// TIA Portal V17 export
// export: Created 2021-12-03T08:13:01.9644948Z, ExportSetting WithDefaults, DisplayName Totally Integrated Automation Portal, DisplayVersion V17, DisplayName TIA Portal Openness, DisplayVersion V17, DisplayName TIA Portal Version Control Interface, DisplayVersion V17, DisplayName STEP 7 Professional, DisplayVersion V17, DisplayName STEP 7 Safety, DisplayVersion V17, DisplayName WinCC Advanced, DisplayVersion V17
FUNCTION_BLOCK "FB_MN_Acc_Ctrl"   // FB61, FBD
VERSION : 0.1
// stored: AutoNumber false, IsIECCheckEnabled true, UDAEnableTagReadback false
   VAR_INPUT
      I_InitTrue { ExternalVisible := 'False'; ExternalWritable := 'False'} : Bool;   // Инициализация
      I_Acc_PwrOnRq { ExternalVisible := 'False'; ExternalWritable := 'False'} : Bool;   // Запрос на включение
      I_AccChil_PwrIsOn { ExternalVisible := 'False'; ExternalWritable := 'False'} : Bool;   // Чиллер включен
      I_Mod220V_PwrIsOn { ExternalVisible := 'False'; ExternalWritable := 'False'} : Bool;   // Модулятор 220 В включен
      I_Mod380V_PwrIsOn { ExternalVisible := 'False'; ExternalWritable := 'False'} : Bool;   // Модулятор 380 В включен
      I_AccCS_PrwIsOn { ExternalVisible := 'False'; ExternalWritable := 'False'} : Bool;   // Ускоритель включен
      I_AccRemMode { ExternalVisible := 'False'; ExternalWritable := 'False'} : Bool;   // Удаленный режим
      I_AccWarmUp { ExternalVisible := 'False'; ExternalWritable := 'False'} : Bool;   // Прогрев ускорителя
      I_AccClear { ExternalVisible := 'False'; ExternalWritable := 'False'} : Bool;   // Предварительная готовность
      I_AccStandby { ExternalVisible := 'False'; ExternalWritable := 'False'} : Bool;   // Пауза
      I_AccReady { ExternalVisible := 'False'; ExternalWritable := 'False'} : Bool;   // Основная готовность
      I_RFOn_Rq { ExternalVisible := 'False'; ExternalWritable := 'False'} : Bool;
      I_XRay_Rq { ExternalVisible := 'False'; ExternalWritable := 'False'} : Bool;
      I_Acc_PwrOffRq { ExternalVisible := 'False'; ExternalWritable := 'False'} : Bool;   // Запрос на отключение
      I_ChillOffDly { ExternalVisible := 'False'; ExternalWritable := 'False'} : Bool;   // Чиллер включен
      I_AccFault { ExternalVisible := 'False'; ExternalWritable := 'False'} : Bool;   // Ошибка ускорителя
      I_NOEStop { ExternalVisible := 'False'; ExternalWritable := 'False'} : Bool;   // Аварийный останов
      I_FltRst { ExternalVisible := 'False'; ExternalWritable := 'False'} : Bool;   // Сигнал сбросить ошибки
      I_FullWarmUp { ExternalVisible := 'False'; ExternalWritable := 'False'} : Bool;   // Полный прогрев
      I_SafePeriIsCls { ExternalVisible := 'False'; ExternalWritable := 'False'} : Bool;   // Периметр закрыт
      I_PwrRst { ExternalVisible := 'False'; ExternalWritable := 'False'} : Bool;
   END_VAR
   VAR_OUTPUT
      O_AccPreh_PwrOn { ExternalVisible := 'False'; ExternalWritable := 'False'} : Bool;   // Включение сушки ускорителя
      O_Mod380V_RlyOn { ExternalVisible := 'False'; ExternalWritable := 'False'} : Bool;   // Включить модулятор 380 В
      O_AccMod220V_PwrOn { ExternalVisible := 'False'; ExternalWritable := 'False'} : Bool;   // Включить модулятор 220 В
      O_Chil_PwrOn { ExternalVisible := 'False'; ExternalWritable := 'False'} : Bool;   // Включить - отключть чиллер
      O_FltRst { ExternalVisible := 'False'; ExternalWritable := 'False'} : Bool;   // Сброс ошибки / Reset
      O_WarmUp { ExternalVisible := 'False'; ExternalWritable := 'False'} : Bool;   // Запрос на прогрев
      O_RFOn { ExternalVisible := 'False'; ExternalWritable := 'False'} : Bool;   // Включить СВЧ
      O_XRay_On { ExternalVisible := 'False'; ExternalWritable := 'False'} : Bool;   // Включить ТИ
      O_FullWarmUp_Rq { ExternalVisible := 'False'; ExternalWritable := 'False'} : Bool;   // Запрос на полный прогрев
      O_Acc_ActState { ExternalVisible := 'False'; ExternalWritable := 'False'} : Int;   // Состояние ускорителя
   END_VAR
   VAR DB_SPECIFIC
      S_PwrRst { ExternalVisible := 'False'} : Bool;
      AxSR { ExternalVisible := 'False'; ExternalWritable := 'False'} : Struct
         Acc230V_PwrOn { ExternalVisible := 'False'; ExternalWritable := 'False'} : Bool;
      END_STRUCT;
      S_Transit { ExternalVisible := 'False'; ExternalWritable := 'False'} : Struct
         InitTrue { ExternalVisible := 'False'; ExternalWritable := 'False'} : Bool;   // Инициализация
         ReqAccPwrOn { ExternalVisible := 'False'; ExternalWritable := 'False'} : Bool;   // Запрос на включение
         ChillOnDly { ExternalVisible := 'False'; ExternalWritable := 'False'} : Bool;   // Чиллер включен
         ModOnDly { ExternalVisible := 'False'; ExternalWritable := 'False'} : Bool;   // Модулятор включен
         AccPrwOn { ExternalVisible := 'False'; ExternalWritable := 'False'} : Bool;   // Ускоритель включен
         NAccPrwOn { ExternalVisible := 'False'; ExternalWritable := 'False'} : Bool;   // Ускоритель НЕ включен
         AccRemMode { ExternalVisible := 'False'; ExternalWritable := 'False'} : Bool;   // Удаленный режим
         NAccRemMode { ExternalVisible := 'False'; ExternalWritable := 'False'} : Bool;   // Местный режим
         AccWarmUp { ExternalVisible := 'False'; ExternalWritable := 'False'} : Bool;   // Прогрев ускорителя
         AccClear { ExternalVisible := 'False'; ExternalWritable := 'False'} : Bool;   // Предварительная готовность
         AccStandby { ExternalVisible := 'False'; ExternalWritable := 'False'} : Bool;   // Пауза
         AccReady { ExternalVisible := 'False'; ExternalWritable := 'False'} : Bool;   // Основная готовность
         AccRfOn { ExternalVisible := 'False'; ExternalWritable := 'False'} : Bool;   // СВЧ включено
         AccRfOff { ExternalVisible := 'False'; ExternalWritable := 'False'} : Bool;
         AccXrayOn { ExternalVisible := 'False'; ExternalWritable := 'False'} : Bool;   // ТИ включено
         AccXrayOff { ExternalVisible := 'False'; ExternalWritable := 'False'} : Bool;   // ТИ вЫключено
         ReqAccPwrOff { ExternalVisible := 'False'; ExternalWritable := 'False'} : Bool;   // Запрос на отключение
         AccNotActive { ExternalVisible := 'False'; ExternalWritable := 'False'} : Bool;   // Ускоритель неактивен
         XrayHeadOffDly { ExternalVisible := 'False'; ExternalWritable := 'False'} : Bool;   // Накал выключен
         ModOffDly { ExternalVisible := 'False'; ExternalWritable := 'False'} : Bool;   // Модулятор выключен
         ChillOffDly { ExternalVisible := 'False'; ExternalWritable := 'False'} : Bool;   // Чиллер включен
         AccFault { ExternalVisible := 'False'; ExternalWritable := 'False'} : Bool;   // Ошибка ускорителя
         ACK_AccFault { ExternalVisible := 'False'; ExternalWritable := 'False'} : Bool;   // Ошибка сброшена
         EStop { ExternalVisible := 'False'; ExternalWritable := 'False'} : Bool;   // Аварийный останов
      END_STRUCT;
   END_VAR
   VAR
      DI_Acc_StateCase { ExternalVisible := 'False'; S7_SetPoint := 'True'} : "FB_Acc_StateCase";
   END_VAR
   VAR DB_SPECIFIC
      S_Acc_ActState { ExternalVisible := 'False'; ExternalWritable := 'False'} : Int;   // Состояние ускорителя
   END_VAR
   VAR_TEMP
      T_Mod230V_PwrOn : Bool;
      T_FltRst : Bool;
      T_Acc230V_PwrOn : Bool;
      T_Mod400V_PwrOn : Bool;
      T_StandBy : Bool;
      T_RFOn : Bool;
      T_XRayOn : Bool;
      T_ReqPwrOn : Bool;
   END_VAR
BEGIN

REGION Network 2: INIT / Инициализация
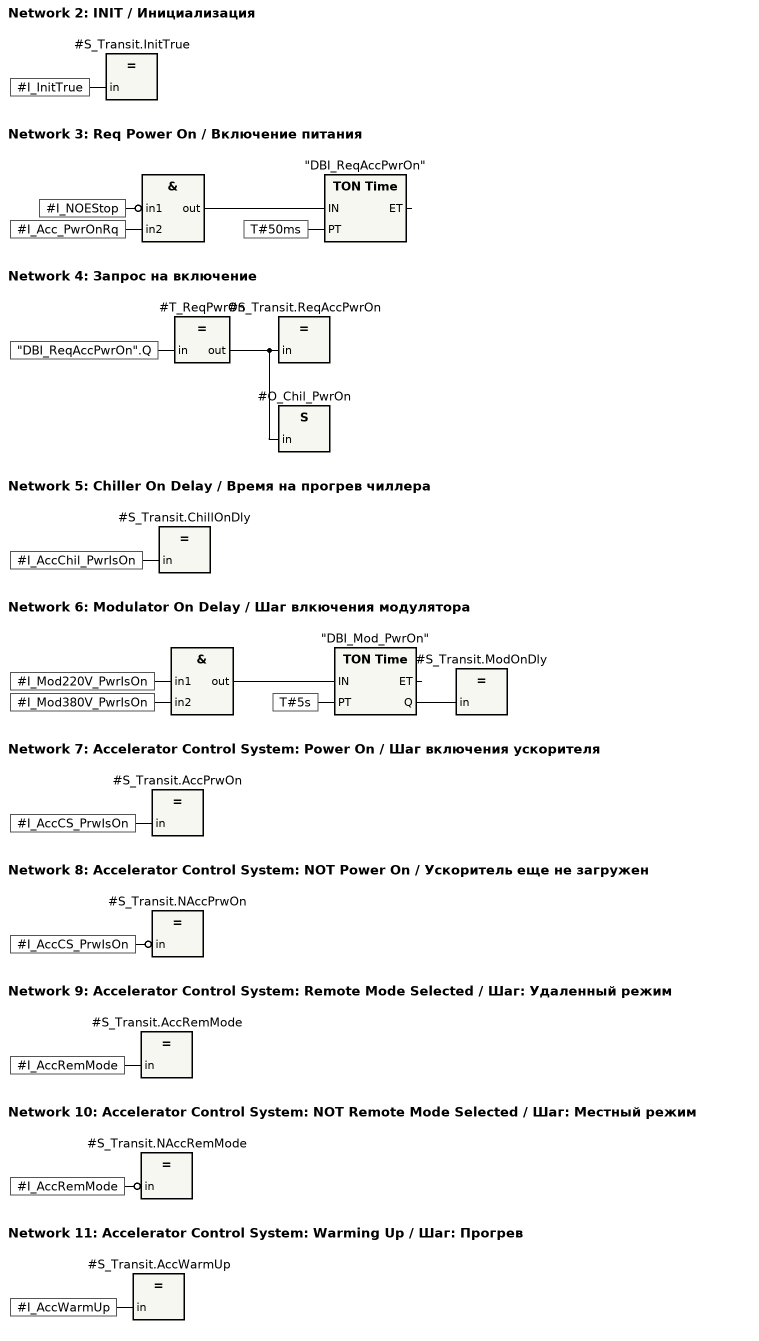
   #S_Transit.InitTrue := #I_InitTrue;
END_REGION

REGION Network 3: Req Power On / Включение питания
   "DBI_ReqAccPwrOn".TON(IN := NOT #I_NOEStop AND #I_Acc_PwrOnRq, PT := T#50ms);
END_REGION

REGION Network 4: Запрос на включение
   #T_ReqPwrOn := "DBI_ReqAccPwrOn".Q;
   #S_Transit.ReqAccPwrOn := "DBI_ReqAccPwrOn".Q;
   IF "DBI_ReqAccPwrOn".Q THEN #O_Chil_PwrOn := TRUE; END_IF;
END_REGION

REGION Network 5: Chiller On Delay / Время на прогрев чиллера
   #S_Transit.ChillOnDly := #I_AccChil_PwrIsOn;
END_REGION

REGION Network 6: Modulator On Delay / Шаг влкючения модулятора
   "DBI_Mod_PwrOn".TON(IN := #I_Mod220V_PwrIsOn AND #I_Mod380V_PwrIsOn, PT := T#5s);
   #S_Transit.ModOnDly := "DBI_Mod_PwrOn".Q;
END_REGION

REGION Network 7: Accelerator Control System: Power On / Шаг включения ускорителя
   #S_Transit.AccPrwOn := #I_AccCS_PrwIsOn;
END_REGION

REGION Network 8: Accelerator Control System: NOT Power On / Ускоритель еще не загружен
   #S_Transit.NAccPrwOn := NOT #I_AccCS_PrwIsOn;
END_REGION

REGION Network 9: Accelerator Control System: Remote Mode Selected / Шаг: Удаленный режим
   #S_Transit.AccRemMode := #I_AccRemMode;
END_REGION

REGION Network 10: Accelerator Control System: NOT Remote Mode Selected / Шаг: Местный режим
   #S_Transit.NAccRemMode := NOT #I_AccRemMode;
END_REGION

REGION Network 11: Accelerator Control System: Warming Up / Шаг: Прогрев
   #S_Transit.AccWarmUp := #I_AccWarmUp;
END_REGION

REGION Network 12: Accelerator Control System: Clear / Шаг: Предварительная готовность
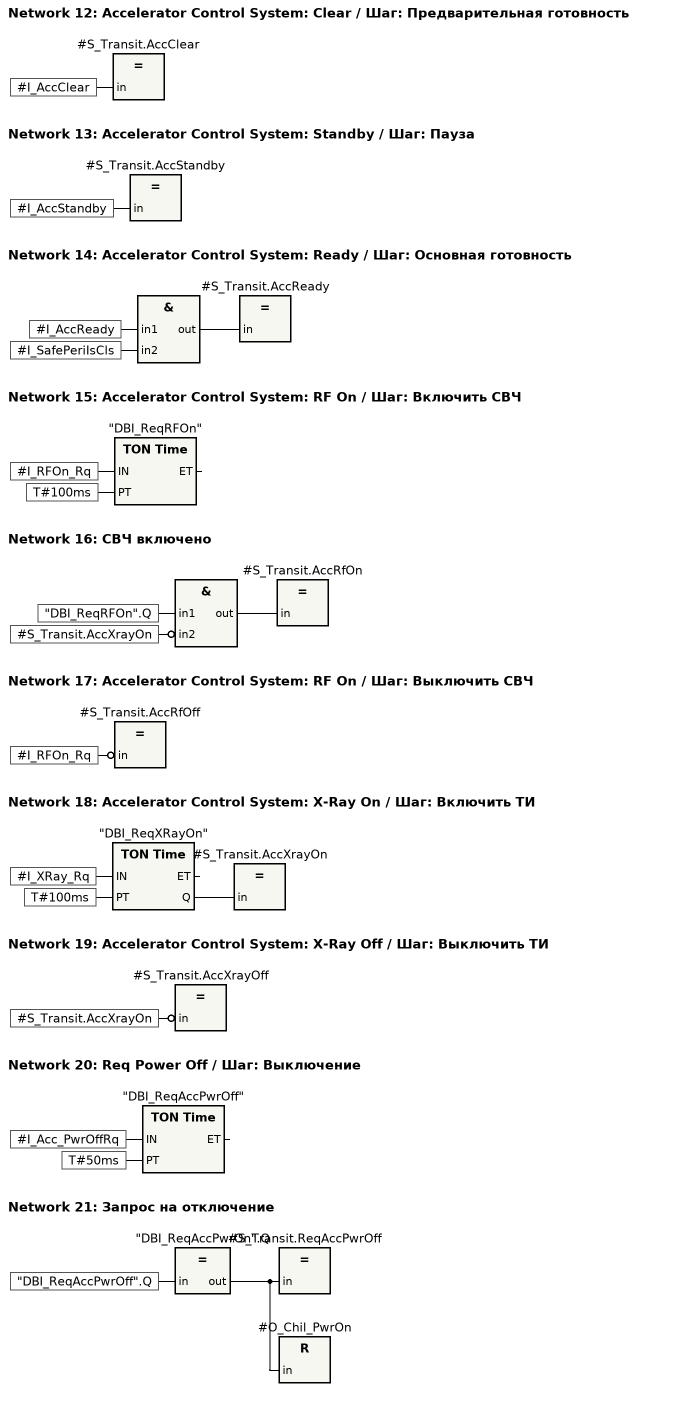
   #S_Transit.AccClear := #I_AccClear;
END_REGION

REGION Network 13: Accelerator Control System: Standby / Шаг: Пауза
   #S_Transit.AccStandby := #I_AccStandby;
END_REGION

REGION Network 14: Accelerator Control System: Ready / Шаг: Основная готовность
   #S_Transit.AccReady := #I_AccReady AND #I_SafePeriIsCls;
END_REGION

REGION Network 15: Accelerator Control System: RF On / Шаг: Включить СВЧ
   "DBI_ReqRFOn".TON(IN := #I_RFOn_Rq, PT := T#100ms);
END_REGION

REGION Network 16: СВЧ включено
   #S_Transit.AccRfOn := "DBI_ReqRFOn".Q AND NOT #S_Transit.AccXrayOn;
END_REGION

REGION Network 17: Accelerator Control System: RF On / Шаг: Выключить СВЧ
   #S_Transit.AccRfOff := NOT #I_RFOn_Rq;
END_REGION

REGION Network 18: Accelerator Control System: X-Ray On / Шаг: Включить ТИ
   "DBI_ReqXRayOn".TON(IN := #I_XRay_Rq, PT := T#100ms);
   #S_Transit.AccXrayOn := "DBI_ReqXRayOn".Q;
END_REGION

REGION Network 19: Accelerator Control System: X-Ray Off / Шаг: Выключить ТИ
   #S_Transit.AccXrayOff := NOT #S_Transit.AccXrayOn;
END_REGION

REGION Network 20: Req Power Off / Шаг: Выключение
   "DBI_ReqAccPwrOff".TON(IN := #I_Acc_PwrOffRq, PT := T#50ms);
END_REGION

REGION Network 21: Запрос на отключение
   "DBI_ReqAccPwrOn".Q := "DBI_ReqAccPwrOff".Q;
   #S_Transit.ReqAccPwrOff := "DBI_ReqAccPwrOff".Q;
   IF "DBI_ReqAccPwrOff".Q THEN #O_Chil_PwrOn := FALSE; END_IF;
END_REGION

REGION Network 22: Accelerator Control System: NOT Clear, Ready, Warming Up / Шаг: ускоритель не активен (снятие накала)
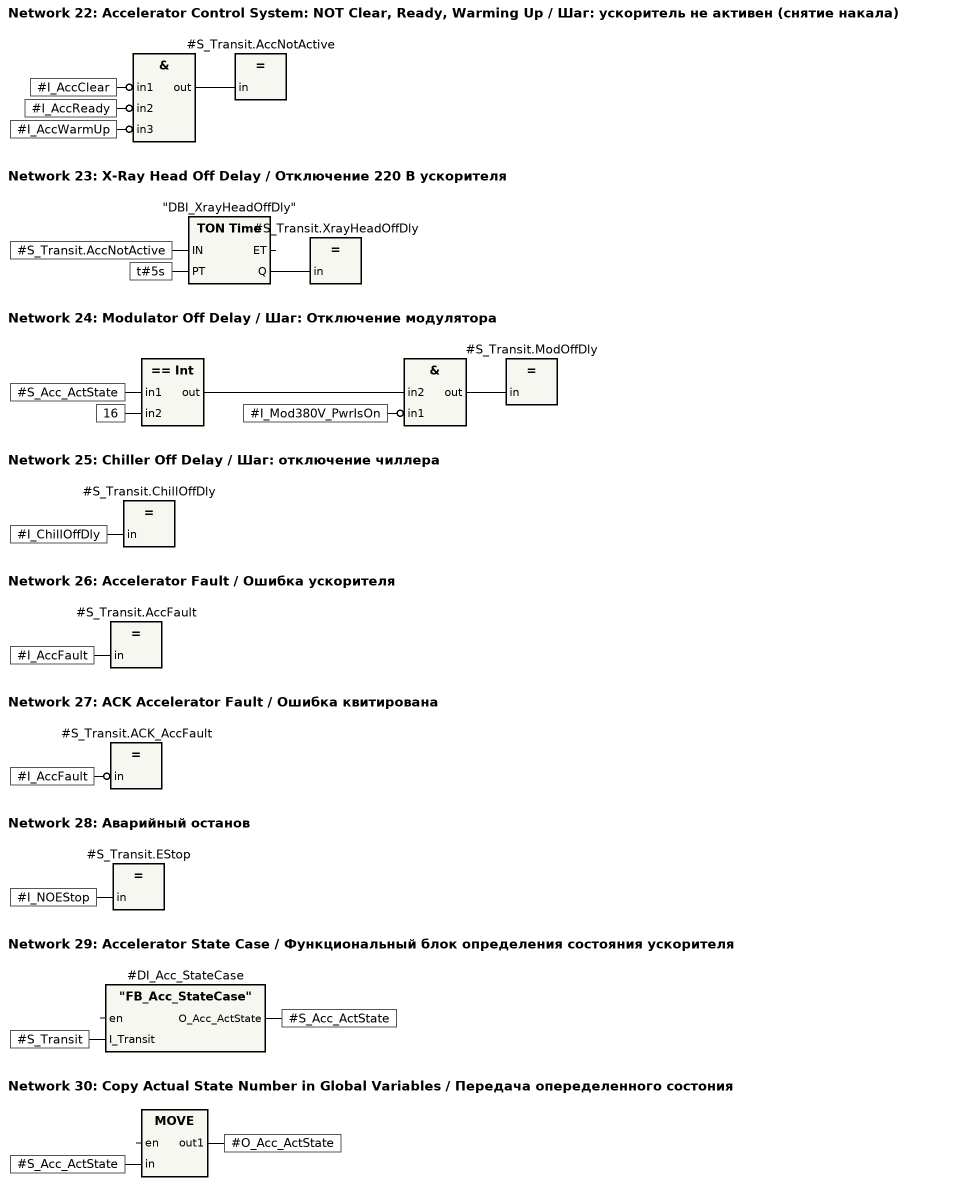
   #S_Transit.AccNotActive := NOT #I_AccClear AND NOT #I_AccReady AND NOT #I_AccWarmUp;
END_REGION

REGION Network 23: X-Ray Head Off Delay / Отключение 220 В ускорителя
   "DBI_XrayHeadOffDly".TON(IN := #S_Transit.AccNotActive, PT := t#5s);
   #S_Transit.XrayHeadOffDly := "DBI_XrayHeadOffDly".Q;
END_REGION

REGION Network 24: Modulator Off Delay / Шаг: Отключение модулятора
   #S_Transit.ModOffDly := (#S_Acc_ActState = 16) AND NOT #I_Mod380V_PwrIsOn;
END_REGION

REGION Network 25: Chiller Off Delay / Шаг: отключение чиллера
   #S_Transit.ChillOffDly := #I_ChillOffDly;
END_REGION

REGION Network 26: Accelerator Fault / Ошибка ускорителя
   #S_Transit.AccFault := #I_AccFault;
END_REGION

REGION Network 27: ACK Accelerator Fault / Ошибка квитирована
   #S_Transit.ACK_AccFault := NOT #I_AccFault;
END_REGION

REGION Network 28: Аварийный останов
   #S_Transit.EStop := #I_NOEStop;
END_REGION

REGION Network 29: Accelerator State Case / Функциональный блок определения состояния ускорителя
   #DI_Acc_StateCase(I_Transit := #S_Transit, O_Acc_ActState => #S_Acc_ActState);   // "FB_Acc_StateCase"
END_REGION

REGION Network 30: Copy Actual State Number in Global Variables / Передача опеределенного состония
   #O_Acc_ActState := #S_Acc_ActState;
END_REGION

REGION Network 31: Accelerator State Case: Actions / Функциональный блок действий
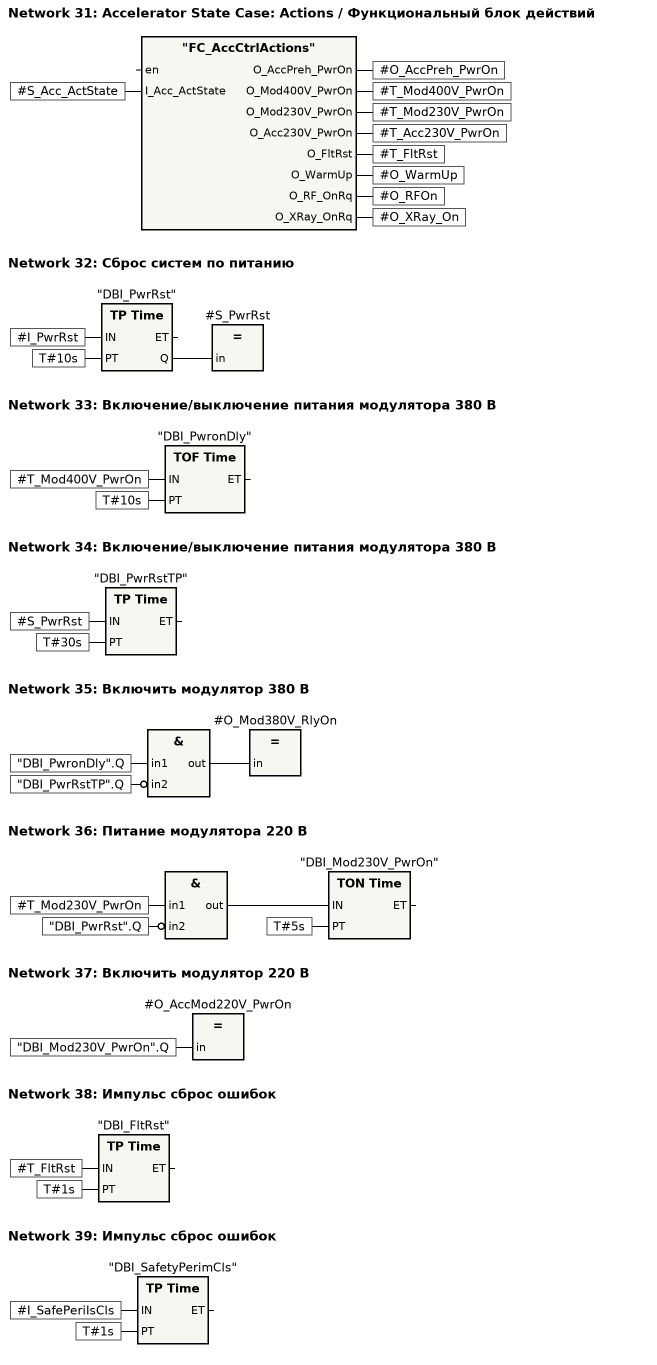
   "FC_AccCtrlActions"(I_Acc_ActState := #S_Acc_ActState,
                       O_AccPreh_PwrOn => #O_AccPreh_PwrOn,
                       O_Mod400V_PwrOn => #T_Mod400V_PwrOn,
                       O_Mod230V_PwrOn => #T_Mod230V_PwrOn,
                       O_Acc230V_PwrOn => #T_Acc230V_PwrOn,
                       O_FltRst => #T_FltRst,
                       O_WarmUp => #O_WarmUp,
                       O_RF_OnRq => #O_RFOn,
                       O_XRay_OnRq => #O_XRay_On);
END_REGION

REGION Network 32: Сброс систем по питанию
   "DBI_PwrRst".TP(IN := #I_PwrRst, PT := T#10s);
   #S_PwrRst := "DBI_PwrRst".Q;
END_REGION

REGION Network 33: Включение/выключение питания модулятора 380 В
   "DBI_PwronDly".TOF(IN := #T_Mod400V_PwrOn, PT := T#10s);
END_REGION

REGION Network 34: Включение/выключение питания модулятора 380 В
   "DBI_PwrRstTP".TP(IN := #S_PwrRst, PT := T#30s);
END_REGION

REGION Network 35: Включить модулятор 380 В
   #O_Mod380V_RlyOn := "DBI_PwronDly".Q AND NOT "DBI_PwrRstTP".Q;
END_REGION

REGION Network 36: Питание модулятора 220 В
   "DBI_Mod230V_PwrOn".TON(IN := #T_Mod230V_PwrOn AND NOT "DBI_PwrRst".Q, PT := T#5s);
END_REGION

REGION Network 37: Включить модулятор 220 В
   #O_AccMod220V_PwrOn := "DBI_Mod230V_PwrOn".Q;
END_REGION

REGION Network 38: Импульс сброс ошибок
   "DBI_FltRst".TP(IN := #T_FltRst, PT := T#1s);
END_REGION

REGION Network 39: Импульс сброс ошибок
   "DBI_SafetyPerimCls".TP(IN := #I_SafePeriIsCls, PT := T#1s);
END_REGION

REGION Network 40: Сброс ошибки
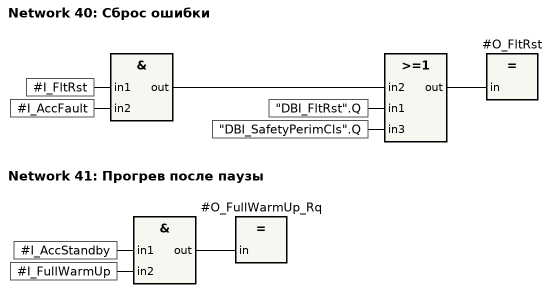
   #O_FltRst := (#I_FltRst AND #I_AccFault) OR "DBI_FltRst".Q OR "DBI_SafetyPerimCls".Q;
END_REGION

REGION Network 41: Прогрев после паузы
   #O_FullWarmUp_Rq := #I_AccStandby AND #I_FullWarmUp;
END_REGION

REGION Network 42: Конец блока
END_REGION
END_FUNCTION_BLOCK
